PROGRAM Proces_2
VAR
	
	Step: INT;
END_VAR

CASE Step OF

0: // wachten op machine aan
IF GVL.Power_ON THEN 
	Step			:=10;
END_IF	


10: // water kan verwarmt worden
GVL.Water_verwarmen := TRUE;

IF GVL.Water_opgewarmt THEN
	Step			:=20;
END_IF

20: // water is opgewarmt. Waneer water niet meer op temperatuur is terug naar step 10
GVL.Water_verwarmen := FALSE;

IF GVL.Water_opgewarmt = FALSE THEN
	Step			:=10;
END_IF
END_CASE

END_PROGRAM

(* stored: Version 1.1.0.1, ProductVersion 3.1.4024.12
   POU Proces_2: Id {8ca36e67-a1d1-4f79-b9da-34b3c20ad082}, SpecialFunc None *)
